(*

.. <legal notes>

legal notes
=================
| SPDX-FileCopyrightText: © 2026 Oleksandr Tiutyk <trofimich@gmail.com>
| SPDX-License-Identifier: LGPL-3.0-only
| For details check: LGPL-3.0-only_

.. _LGPL-3.0-only: https://www.gnu.org/licenses/lgpl-3.0.en.html

.. </legal notes>

*)

FUNCTION_BLOCK ABSTRACT CompositeDevice
VAR_GENERIC CONSTANT
	{attribute 'hide'} 
    _ChildCount : TOF_Core.INT_LENGTH := 0;
END_VAR
EXTENDS BranchAutomationComponent IMPLEMENTS ICompositeDevice
VAR
	{attribute 'hide'} 
	_Parent : IParentAutomationComponent;
END_VAR

METHOD FINAL BubbleEvent
VAR_INPUT
	event : TOF_Core.IEvent;
END_VAR
VAR
	stopPropagation : BOOL;
	
	parentAsBubbleEventDispatcher : TOF_Core.IBubbleEventDispatcher;
END_VAR
OnEventReceived(event := event, stopPropagation => stopPropagation);

IF stopPropagation THEN
	RETURN;
END_IF

IF __QUERYINTERFACE(Parent, parentAsBubbleEventDispatcher) THEN
	parentAsBubbleEventDispatcher.BubbleEvent(event);
END_IF
END_METHOD

{attribute 'monitoring' := 'call'}
PROPERTY FINAL ChildCount : TOF_Core.INT_LENGTH
GET
ChildCount := _ChildCount;
END_GET
END_PROPERTY

{attribute 'monitoring' := 'call'}
PROPERTY ABSTRACT Children : REFERENCE TO ARRAY [0.._ChildCount - 1] OF IChildAutomationComponent
GET
END_GET
END_PROPERTY

METHOD FB_init : BOOL
VAR_INPUT
	(* if TRUE, the retain variables are initialized (warm start / cold start)*)
	bInitRetains	: BOOL;
	(* if TRUE, the instance afterwards gets moved into the copy code (online change)*)
	bInCopyCode	: BOOL;
	name : WSTRING;
	parent : IParentAutomationComponent;
END_VAR
_Parent := parent;
END_METHOD

{attribute 'monitoring' := 'call'}
PROPERTY FINAL Parent : IParentAutomationComponent
GET
Parent := _Parent;
END_GET
END_PROPERTY

METHOD FINAL ProcessInput
VAR
	exceptionCode : __SYSTEM.ExceptionCode;
	exception : TOF_Core.IException;	
	exceptionReaction : TOF_Core.EXCEPTION_REACTION;
	
	childCriticalErrorReaction : CHILD_CRITICAL_ERROR_REACTION;
	
	i : INT;
		
	child : IChildAutomationComponent;	

	inputDevice : IInputLeafAutomationComponent;
END_VAR
__TRY
	OnBeforeDevicesProcessInput();
__CATCH(exceptionCode)		
	exception := TOF_Core.ExceptionManager.GetLastException(exceptionCode);
					
	exceptionReaction := OnHandleException(exception, 'OnBeforeDevicesProcessInput');

	ProcessException(exception, exceptionReaction, "OnBeforeDevicesProcessInput error");
__ENDTRY

FOR i := 0 TO _ChildCount - 1 DO
	child := TryGetChildByIndex(i);

	IF NOT child.Enabled OR_ELSE NOT __QUERYINTERFACE(child, inputDevice) THEN
		CONTINUE;
	END_IF
	
	inputDevice.ProcessInput();

	IF inputDevice.HasError AND_THEN inputDevice.Error.Severity = TOF_Core.ERROR_SEVERITY.CRITICAL THEN
		childCriticalErrorReaction := HandleChildCriticalError(inputDevice);
		
		ProcessChildError(inputDevice.Error, childCriticalErrorReaction, TOF_Core.WideStrings.Concat255("Child[", TO_WSTRING(i), "(", inputDevice.Name, ")].ProcessInput error"));
	END_IF		
END_FOR

__TRY
	OnAfterDevicesProcessInput();
__CATCH(exceptionCode)		
	exception := TOF_Core.ExceptionManager.GetLastException(exceptionCode);
					
	exceptionReaction := OnHandleException(exception, 'OnAfterDevicesProcessInput');

	ProcessException(exception, exceptionReaction, "OnAfterDevicesProcessInput error");
__ENDTRY
END_METHOD

METHOD FINAL ProcessOutput
VAR
	exceptionCode : __SYSTEM.ExceptionCode;
	exception : TOF_Core.IException;	
	exceptionReaction : TOF_Core.EXCEPTION_REACTION;
	
	childCriticalErrorReaction : CHILD_CRITICAL_ERROR_REACTION;
	
	i : INT;
		
	child : IChildAutomationComponent;	

	outputDevice : IOutputLeafAutomationComponent;
END_VAR
__TRY
	OnBeforeDevicesProcessOutput();
__CATCH(exceptionCode)		
	exception := TOF_Core.ExceptionManager.GetLastException(exceptionCode);
					
	exceptionReaction := OnHandleException(exception, 'OnBeforeDevicesProcessOutput');

	ProcessException(exception, exceptionReaction, "OnBeforeDevicesProcessOutput error");
__ENDTRY

FOR i := 0 TO _ChildCount - 1 DO
	child := TryGetChildByIndex(i);

	IF NOT child.Enabled OR_ELSE NOT __QUERYINTERFACE(child, outputDevice) THEN
		CONTINUE;
	END_IF
	
	outputDevice.ProcessOutput();
	
	IF outputDevice.HasError AND_THEN outputDevice.Error.Severity = TOF_Core.ERROR_SEVERITY.CRITICAL THEN
		childCriticalErrorReaction := HandleChildCriticalError(outputDevice);
		
		ProcessChildError(outputDevice.Error, childCriticalErrorReaction, TOF_Core.WideStrings.Concat255("Child[", TO_WSTRING(i), "(", outputDevice.Name, ")].ProcessOutput error"));
	END_IF
END_FOR

__TRY
	OnAfterDevicesProcessOutput();
__CATCH(exceptionCode)		
	exception := TOF_Core.ExceptionManager.GetLastException(exceptionCode);
					
	exceptionReaction := OnHandleException(exception, 'OnAfterDevicesProcessOutput');

	ProcessException(exception, exceptionReaction, "OnAfterDevicesProcessOutput error");
__ENDTRY
END_METHOD

METHOD FINAL TryGetChildByIndex : IChildAutomationComponent
VAR_INPUT
	index : TOF_Core.INT_INDEX;
END_VAR
IF __ISVALIDREF(Children) AND_THEN index >= 0 AND_THEN index <= _ChildCount THEN
	TryGetChildByIndex := Children[index];
END_IF
END_METHOD

METHOD PROTECTED FINAL Validate
VAR
	notSpecifiedException : TOF_Core.DataMemberNotSpecifiedException;
END_VAR
IF _Parent = 0 THEN
	notSpecifiedException.ThrowByObject(THIS^, __POUNAME(), __POSITION(), 'Parent');						
END_IF

IF ChildCount > 0 AND_THEN NOT __ISVALIDREF(Children) THEN
	notSpecifiedException.ThrowByObject(THIS^, __POUNAME(), __POSITION(), 'Children');
END_IF
END_METHOD

END_FUNCTION_BLOCK

(* stored: Version 1.1.0.1
   POU CompositeDevice: Id {25bfda0d-9225-4be2-8314-f8314e830df8}, SpecialFunc None
   Folder Overriden methods: Id {8e7fddf3-79b8-4a8a-9258-2efb57fe9a7d}
   Method BubbleEvent: Id {ec63c85f-f731-4851-bd8e-f85a62e07837}
   Property ChildCount: Id {eab6dfe5-2f53-4cc8-87ce-0fc821a75f9c}
   Get Get: Id {46ef8b88-c91b-4061-8848-8d8aa1c34fff}
   Property Children: Id {5eb8cc14-af21-41a6-964e-854d2107c6da}
   Get Get: Id {92c9163e-e171-4a3b-8e8e-5251e6af78eb}
   Method FB_init: Id {515605cc-0879-42b7-b0de-34f0ad85bef8}
   Property Parent: Id {8abf624b-c9ed-4996-8788-b464b8e15520}
   Get Get: Id {872e7375-00a6-46e3-b1e4-754a1ea8aef4}
   Method ProcessInput: Id {169f608c-73af-42d0-b266-fd32baea3032}
   Method ProcessOutput: Id {d8822de7-f12d-43fe-bdcd-3812e5246f80}
   Method TryGetChildByIndex: Id {d6468cc2-d65d-413d-b788-a326d0027f11}
   Method Validate: Id {cbb4acd1-d175-4a92-bf2b-4e4a64c68356} *)
